KUKA KRL program: stiffness.src, stiffness.dat

--- stiffness.src ---
&ACCESS RVP
&REL 23
&PARAM TEMPLATE = C:\KRC\Roboter\Template\vorgabe
&PARAM EDITMASK = *
DEF stiffness( )

DECL STIFFNESS customStiffness
;FOLD INI

  ;FOLD BASISTECH INI
    GLOBAL INTERRUPT DECL 3 WHEN $STOPMESS==TRUE DO IR_STOPM ( )
    INTERRUPT ON 3
    BAS (#INITMOV,0 )
  ;ENDFOLD (BASISTECH INI)
;FOLD SPOTTECH INI
;USERSPOT(#INIT)
;ENDFOLD (SPOTTECH INI)
;FOLD GRIPPERTECH INI
;USER_GRP(0,DUMMY,DUMMY,GDEFAULT)
;ENDFOLD (GRIPPERTECH INI)
  ;FOLD USER INI
    ;Make your modifications here

  ;ENDFOLD (USER INI)
;ENDFOLD (INI)

;Start in control position mode
$STIFFNESS.STRATEGY=10
$OV_PRO=75
;FOLD PTP StartPos  Vel= 100 % PDAT3 Tool[2] Base[0]
$BWDSTART = FALSE
PDAT_ACT=PPDAT3
FDAT_ACT=FStartPos
BAS(#PTP_PARAMS,100)
PTP XStartPos
;ENDFOLD

HALT
;Free XYZ RXRYRZ

customStiffness=$STIFFNESS
customStiffness.STRATEGY=20 ;Cartesian Impedance control
customStiffness.FRAMETYPE=#TOOL
customStiffness.TOOL=TOOL_DATA[2] ;Force sensor as tool
customStiffness.CPSTIFFNESS={x 0, y 0, z 0, a 0, b 0, c 0} ;Cartesian stiffness
customStiffness.CPDAMPING={x 0.5, y 0.5, z 0.5, a 0.5, b 0.5, c 0.5} ;Cartesian damping
customStiffness.AXISSTIFFNESS={a1 0,a2 0, a3 0, a4 0, a5 0, a6 0, e1 0} ;Axis stiffness
customStiffness.CPMAXDELTA={x 1399.0, y 1399.0, z 1399.0, a 1399.0, b 1399.0, c 1399.0}
$STIFFNESS=customStiffness

;FOLD PTP StartPos  Vel= 100 % PDAT3 Tool[2] Base[0]
$BWDSTART = FALSE
PDAT_ACT=PPDAT3
FDAT_ACT=FStartPos
BAS(#PTP_PARAMS,100)
PTP XStartPos
;ENDFOLD

;In FREE XYZ ABC
HALT
;Stiffness no move

customStiffness=$STIFFNESS
customStiffness.STRATEGY=20 ;Cartesian Impedance control
customStiffness.FRAMETYPE=#TOOL
customStiffness.TOOL=TOOL_DATA[2] ;Force sensor as tool
customStiffness.CPSTIFFNESS={x 5000, y 5000, z 5000, a 300, b 300, c 300} ;Cartesian stiffness
customStiffness.CPDAMPING={x 0.5, y 0.5, z 0.5, a 0.5, b 0.5, c 0.5} ;Cartesian damping
customStiffness.AXISSTIFFNESS={a1 500,a2 500, a3 500, a4 500, a5 500, a6 500, e1 500} ;Axis stiffness

customStiffness.CPMAXDELTA={x 1399.0, y 1399.0, z 1399.0, a 1399.0, b 1399.0, c 1399.0}
$STIFFNESS=customStiffness

;FOLD PTP StartPos  Vel= 100 % PDAT3 Tool[2] Base[0]
$BWDSTART = FALSE
PDAT_ACT=PPDAT3
FDAT_ACT=FStartPos
BAS(#PTP_PARAMS,100)
PTP XStartPos
;ENDFOLD

;NO MOVE
HALT
;Z free


customStiffness=$STIFFNESS
customStiffness.STRATEGY=20 ;Cartesian Impedance control
customStiffness.FRAMETYPE=#TOOL
customStiffness.TOOL=TOOL_DATA[2] ;Force sensor as tool
customStiffness.CPSTIFFNESS={x 1000, y 1000, z 0, a 300, b 300, c 300} ;Cartesian stiffness
customStiffness.CPDAMPING={x 0.7, y 0.7, z 0.7, a 0.7, b 0.7, c 0.7} ;Cartesian damping
customStiffness.AXISSTIFFNESS={a1 200,a2 200, a3 200, a4 200, a5 200, a6 200, e1 200} ;Axis stiffness
$STIFFNESS=customStiffness

;FOLD PTP StartPos  Vel= 100 % PDAT3 Tool[2] Base[0]
$BWDSTART = FALSE
PDAT_ACT=PPDAT3
FDAT_ACT=FStartPos
BAS(#PTP_PARAMS,100)
PTP XStartPos
;ENDFOLD

;Z FREE
HALT
;XYZ  free


customStiffness=$STIFFNESS
customStiffness.STRATEGY=20 ;Cartesian Impednace control
customStiffness.FRAMETYPE=#TOOL ;

customStiffness.CPSTIFFNESS={x 0, y 0, z 0, a 300, b 300, c 300} ;Cartesian impedance control
customStiffness.CPDAMPING={x 0.7, y 0.7, z 0.7, a 0.7, b 0.7, c 0.7} ;Cartesian damping
customStiffness.AXISSTIFFNESS={a1 1,a2 200, a3 200, a4 200, a5 200, a6 200, e1 200} ;Axis stiffness
$STIFFNESS=customStiffness

;FOLD PTP StartPos  Vel= 100 % PDAT3 Tool[2] Base[0]
$BWDSTART = FALSE
PDAT_ACT=PPDAT3
FDAT_ACT=FStartPos
BAS(#PTP_PARAMS,100)
PTP XStartPos
;ENDFOLD

;XYZ FREE
HALT
;ABC Free

customStiffness=$STIFFNESS
customStiffness.STRATEGY=20 ;Cartesian Impedance control
customStiffness.FRAMETYPE=#TOOL

customStiffness.CPSTIFFNESS={x 2000, y 2000, z 2000, a 0, b 0, c 0} ;Cartesian stiffness
customStiffness.CPDAMPING={x 0.7, y 0.7, z 0.7, a 0.7, b 0.7, c 0.7} ;Cartesian damping

$STIFFNESS=customStiffness

;FOLD PTP StartPos  Vel= 100 % PDAT8 Tool[1]:Greifer leer Base[0]
$BWDSTART = FALSE
PDAT_ACT=PPDAT8
FDAT_ACT=FStartPos
BAS(#PTP_PARAMS,100)
PTP XStartPos
;ENDFOLD

;ABC FREE
;End script
HALT

END

--- stiffness.dat ---
&ACCESS RVO
&REL 23
&PARAM TEMPLATE = C:\KRC\Roboter\Template\vorgabe
&PARAM EDITMASK = *
DEFDAT stiffness
;FOLD EXTERNAL DECLARATIONS;%{PE}%MKUKATPBASIS,%CEXT,%VCOMMON,%P
;FOLD GRIPPERTECH EXT
;EXT  H50 (INT  :IN,INT  :IN,INT  :IN,GRP_TYP  :IN )
;ENDFOLD (GRIPPERTECH EXT)
;FOLD SPOTTECH EXT
;EXT  USERSPOT (S_COMMAND  :IN,SPOT_TYPE  :IN )
;ENDFOLD (SPOTTECH EXT)
;FOLD BASISTECH EXT;%{PE}%MKUKATPBASIS,%CEXT,%VEXT,%P
EXT  BAS (BAS_COMMAND  :IN,REAL  :IN )
DECL INT SUCCESS
;ENDFOLD (BASISTECH EXT)
;FOLD USER EXT;%{E}%MKUKATPUSER,%CEXT,%VEXT,%P
;Make here your modifications

;ENDFOLD (USER EXT)
;ENDFOLD (EXTERNAL DECLERATIONS)
DECL BASIS_SUGG_T LAST_BASIS={POINT1[] "StartPos                ",POINT2[] "StartPos                ",CP_PARAMS[] "CPDAT0                  ",PTP_PARAMS[] "PDAT10                  ",CONT[] "                        ",CP_VEL[] "2.0                     ",PTP_VEL[] "100                     "}
DECL E6POS XSTARTPOS={X -539.306213,Y 102.192902,Z 288.445496,A -118.0214,B -9.07260182E-05,C 179.411301,S 1,T 37,E1 -10.5886898,E2 0.0,E3 0.0,E4 0.0,E5 0.0,E6 0.0}
DECL FDAT FStartPos={TOOL_NO 2,BASE_NO 0,IPO_FRAME #BASE,POINT2[] " "}
DECL PDAT PPDAT3={VEL 100.0,ACC 100.0,APO_DIST 100.0}
DECL PDAT PPDAT4={VEL 100.0,ACC 100.0,APO_DIST 100.0}
DECL PDAT PPDAT5={VEL 100.0,ACC 100.0,APO_DIST 100.0}
DECL PDAT PPDAT6={VEL 100.0,ACC 100.0,APO_DIST 100.0}
DECL PDAT PPDAT7={VEL 100.0,ACC 100.0,APO_DIST 100.0}
DECL PDAT PPDAT8={VEL 100.0,ACC 100.0,APO_DIST 100.0}
DECL PDAT PPDAT9={VEL 100.0,ACC 100.0,APO_DIST 100.0}
DECL PDAT PPDAT10={VEL 100.0,ACC 100.0,APO_DIST 100.0}
DECL E6POS XProblemPos={X 46.9002914,Y 50.9478912,Z 774.595215,A -95.3028717,B -24.5935307,C 86.300827,S 0,T 37,E1 -9.96122646,E2 0.0,E3 0.0,E4 0.0,E5 0.0,E6 0.0}
DECL FDAT FProblemPos={TOOL_NO 2,BASE_NO 0,IPO_FRAME #BASE,POINT2[] " "}
DECL LDAT LCPDAT1={VEL 2.0,ACC 100.0,APO_DIST 100.0,APO_FAC 50.0,ORI_TYP #VAR}
ENDDAT
